FUNCTION IsInRangeInclusive2D : BOOL
VAR_INPUT
	point : Point2D;
	range : Range2D;
END_VAR

IsInRangeInclusive2D := 
	IsInRangeInclusive(point.X, range.X)
	AND IsInRangeInclusive(point.Y, range.Y)
	;

END_FUNCTION

(* stored: Version 1.1.0.1
   POU IsInRangeInclusive2D: Id {e3369920-1f5c-099b-2b1a-c1f44360d0ba}, SpecialFunc None *)
